FUNCTION_BLOCK FB_FalliblePublic IMPLEMENTS I_FalliblePublic
VAR
    {attribute 'pytmc' := '
        pv: Error
        io: i
        field: DESC TRUE if in error state. FALSE if not.
    '}
    bError : BOOL;
    {attribute 'pytmc' := '
        pv: ErrorMsg
        io: i
        field: DESC Message to aid in debugging if error is true.
    '}
    sErrorMsg : T_MaxString;
END_VAR


METHOD ClearError

bError := FALSE;
sErrorMsg := '';
END_METHOD


METHOD PUBLIC GetError : BOOL

GetError := bError;
END_METHOD


METHOD PUBLIC GetErrorMsg : T_MaxString

GetErrorMsg := sErrorMsg;
END_METHOD


METHOD SetError
VAR_INPUT
    Msg : T_MaxString;
END_VAR

bError := TRUE;
sErrorMsg := Msg;
END_METHOD

END_FUNCTION_BLOCK

(* stored: Version 1.1.0.1
   POU FB_FalliblePublic: Id {b31e2ad8-b7ee-4d66-a0d2-490aab45eadc}, SpecialFunc None
   Method ClearError: Id {e508f329-7528-441e-8224-c35c1c1d76fc}
   Method GetError: Id {9e2f6e28-2861-47e9-a8e4-2a94f8af3a74}
   Method GetErrorMsg: Id {6d3edd89-1b7c-4e6d-b76c-799a48331a0a}
   Method SetError: Id {c14920fb-6747-422b-8d39-c0e873f896ca} *)
